FUNCTION_BLOCK FB_StateClosed
VAR_IN_OUT
	stAxis  	: ARRAY [GVL.cXP .. GVL.cXM] OF ST_AxisGroup;	
	bTopEntry	: BOOL;
	nRet	: INT;
	nExt	: INT;
END_VAR

VAR
	nCurrentState	: INT;
	nNextState		: INT;
END_VAR



IF bTopEntry = TRUE THEN
	bTopEntry := FALSE;
	nRet := 1 - nRet;
	nExt := 1 - nExt;
	nNextState := 1000;
END_IF	
nCurrentState := nNextState;

CASE nCurrentState OF

	1000:


END_CASE

END_FUNCTION_BLOCK

(* stored: Version 1.1.0.1, ProductVersion 3.1.4020.12
   POU FB_StateClosed: Id {c84953d7-64f8-44ca-8f15-641427cb62d6}, SpecialFunc None *)
